{attribute 'GeneratedUsingTerminal: KL2531-0001'}
{attribute addProperty BoxType "KL2531-0001"}
{attribute addProperty Id "StatusAT %I*USINT0PositionAT %I*UDINT0ExtStatusAT %I*UINT0CtrlAT %Q*USINT0VelocityAT %Q*DINT0ExtCtrlAT %Q*UINT0"}
{attribute addProperty CRC "219752944"}
{attribute addProperty Size "0"}
TYPE Channel_0D1929F0 :
STRUCT
	{attribute addProperty Name "Status"}
	Status AT %I* : USINT;
	{attribute addProperty Name "Position"}
	Position AT %I* : UDINT;
	{attribute addProperty Name "ExtStatus"}
	ExtStatus AT %I* : UINT;
	{attribute addProperty Name "Ctrl"}
	Ctrl AT %Q* : USINT;
	{attribute addProperty Name "Velocity"}
	Velocity AT %Q* : DINT;
	{attribute addProperty Name "ExtCtrl"}
	ExtCtrl AT %Q* : UINT;
END_STRUCT
END_TYPE

(* stored: Version 1.2.0.0, ProductVersion 3.1.4024.11
   DUT Channel_0D1929F0: Id {382f727e-85d5-4342-aa4c-51a6eb2f2f82} *)
